Yaskawa INFORM job: TCP_LONG_SPIKE.JBI

/JOB
//NAME TCP_LONG_SPIKE
///FOLDERNAME INNE
//POS
///NPOS 19,19,0,0,0,0
///TOOL 0
///POSTYPE PULSE
///PULSE
C00000=1438,-26317,27906,8736,106372,51369
C00001=22519,18670,87499,5940,107841,50333
C00002=72045,-24864,32574,-1560,104707,59890
C00003=108333,-42111,16594,-4633,100550,61937
C00004=134499,-61344,-139,-4585,95189,58754
C00005=181776,-66405,-487,-2155,95408,54976
C00006=-177680,-78687,-9825,11776,89737,59107
C00007=-94004,-51797,7976,15111,97265,64663
C00008=-38822,-38996,15704,10214,99595,70826
C00009=-3174,-42247,10064,7228,99414,64383
C00010=-25156,-62829,-8742,11339,93683,54123
C00011=56785,-71763,-15900,1594,91823,44302
C00012=105925,-62603,-4250,-3996,101527,26323
C00013=208951,-65131,2494,562,102070,32584
C00014=-85350,-61139,-2104,16493,100743,33671
C00015=-172828,-64866,2332,13638,100586,38470
C00016=-221612,-80134,-9838,7558,94693,38505
C00017=-161099,-109519,-30953,15018,75130,40688
C00018=56898,-86482,-26184,1498,82657,47475
BC00000=260759,1064965,689025
BC00001=260759,1064965,689025
BC00002=260759,1064966,689015
BC00003=260759,1064966,689015
BC00004=260759,1064966,689015
BC00005=260759,1064967,689007
BC00006=260759,1064967,689007
BC00007=260759,1064967,689004
BC00008=260759,1064967,689004
BC00009=260759,1064967,689004
BC00010=260759,1064967,689004
BC00011=260759,1064967,688996
BC00012=260759,1064967,688996
BC00013=260759,1064967,688994
BC00014=260759,1064967,688994
BC00015=260759,1064967,688994
BC00016=260759,1064967,688994
BC00017=260759,1064967,688994
BC00018=260759,1064967,688992
//INST
///DATE 2023/10/04 15:12
///ATTR SC,RW
///GROUP1 RB1,BS1
NOP
MOVJ C00000 BC00000 VJ=0.78
MOVJ C00001 BC00001 VJ=0.78
MOVJ C00002 BC00002 VJ=0.78
MOVJ C00003 BC00003 VJ=0.78
MOVJ C00004 BC00004 VJ=0.78
MOVJ C00005 BC00005 VJ=0.78
MOVJ C00006 BC00006 VJ=0.78
MOVJ C00007 BC00007 VJ=0.78
MOVJ C00008 BC00008 VJ=0.78
MOVJ C00009 BC00009 VJ=0.78
MOVJ C00010 BC00010 VJ=0.78
MOVJ C00011 BC00011 VJ=0.78
MOVJ C00012 BC00012 VJ=0.78
MOVJ C00013 BC00013 VJ=0.78
MOVJ C00014 BC00014 VJ=0.78
MOVJ C00015 BC00015 VJ=0.78
MOVJ C00016 BC00016 VJ=0.78
MOVJ C00017 BC00017 VJ=0.78
MOVJ C00018 BC00018 VJ=0.78
END
